// LS Electric XG5000 project: 25.04.03_프로젝트2_컨베이어제어
// PLC LSPLC

PROGRAM NewProgram (task: 스캔 프로그램)

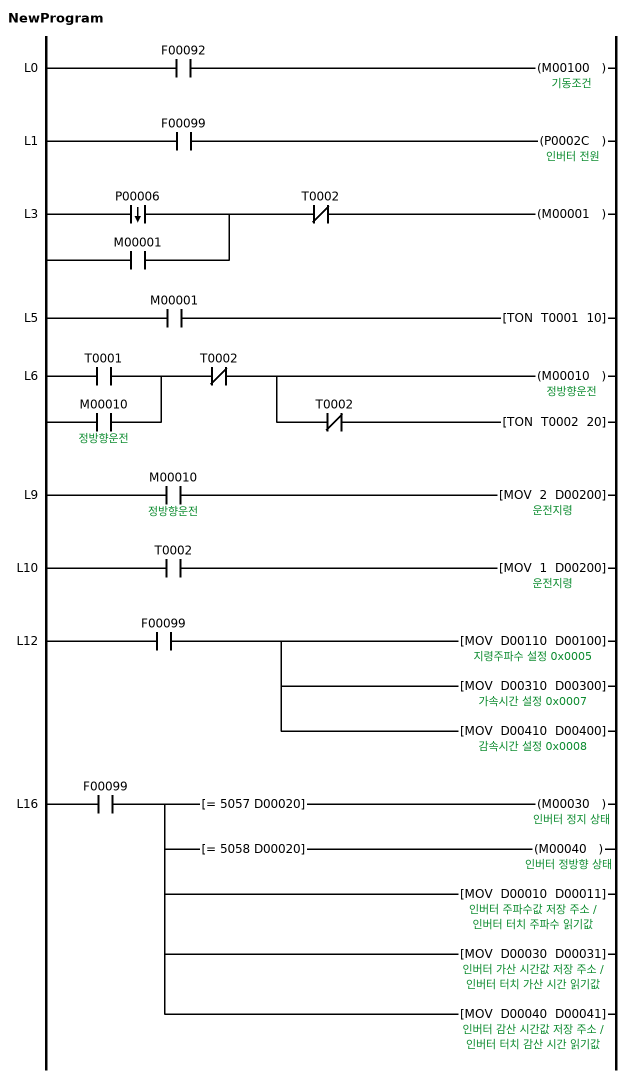
; L0
LOAD      F00092
OUT       M00100	// 기동조건
; L1
LOAD      F00099
OUT       P0002C	// 인버터 전원
; L3
LOADN     P00006
OR        M00001
AND NOT   T0002
OUT       M00001
; L5
LOAD      M00001
TON       T0001 10
; L6
LOAD      T0001
OR        M00010	// 정방향운전
AND NOT   T0002
OUT       M00010	// 정방향운전
AND NOT   T0002
TON       T0002 20
; L9
LOAD      M00010	// 정방향운전
MOV       2 D00200	// 운전지령
; L10
LOAD      T0002
MOV       1 D00200	// 운전지령
; L12
LOAD      F00099
MOV       D00110 D00100	// 지령주파수 설정 0x0005
MOV       D00310 D00300	// 가속시간 설정 0x0007
MOV       D00410 D00400	// 감속시간 설정 0x0008
; L16
LOAD      F00099
MPUSH
AND=      5057 D00020
OUT       M00030	// 인버터 정지 상태
MLOAD
AND=      5058 D00020
OUT       M00040	// 인버터 정방향 상태
MPOP
MOV       D00010 D00011	// 인버터 주파수값 저장 주소 / 인버터 터치 주파수 읽기값
MOV       D00030 D00031	// 인버터 가산 시간값 저장 주소 / 인버터 터치 가산 시간 읽기값
MOV       D00040 D00041	// 인버터 감산 시간값 저장 주소 / 인버터 터치 감산 시간 읽기값

VARIABLES AND COMMENTS (devices not used above)
M00002	BIT	정지
M00020	BIT	역방향운전
M00050	BIT	인버터 역방향 상태